DATA_BLOCK "LMB_ModbusDeviceRtu_DataDb"
{ S7_Optimized_Access := 'FALSE' }
VERSION : 0.1
NON_RETAIN
   STRUCT
      buffer : Array[0..125] of Word;
      writeBuffer : Array[0..125] of Word;
   END_STRUCT;


BEGIN

END_DATA_BLOCK

